FUNCTION_BLOCK fbInfluxPerformanceLogging
VAR
	{attribute clr [ReadOnly()]}
	{attribute clr [CompilerOmits("BuilderPlainer")]}
	{attribute clr [RenderIgnore()]}
	_logStart : ULINT;
	{attribute clr [RenderIgnore()]}
	{attribute clr [CompilerOmits("BuilderPlainer")]}
	_logDone : ULINT;
	
	_data : InfluxData;	
END_VAR

_data.CycleCount := TwinCAT_SystemInfoVarList._TaskInfo[1].CycleCount;
_data.CycleTime := TwinCAT_SystemInfoVarList._TaskInfo[1].CycleTime;
_data.LastExecTime := TwinCAT_SystemInfoVarList._TaskInfo[1].LastExecTime;

IF(_logStart <= _logDone) THEN 
	_logStart := _logStart + 1; 
END_IF

END_FUNCTION_BLOCK

(* stored: Version 1.1.0.1, ProductVersion 3.1.4024.3
   POU fbInfluxPerformanceLogging: Id {5ff4b3e5-e813-4ba9-ad4c-d1bedb24728c}, SpecialFunc None *)
